ABB RobotStudio station: TCP_Station.rspag

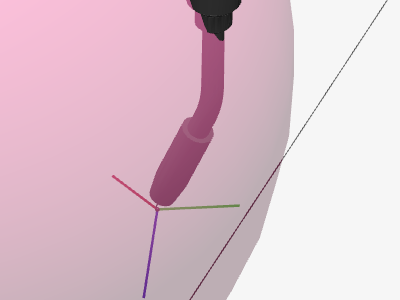
--- station ---
Station TCP_Station (saved by RobotStudio 24.3.10835.0)
Controller IRB2600_12_165, task T_ROB1: task frame (RAPID world) sits at (0, 0, 400) mm in the station
Controller IRB2600_12_165
  mechanical unit ROB_1: IRB2600_12_165_C_01, 6 joints, base frame (0, 0, 0) mm
Layout (positions relative to the parent item):
  - IRB2600_12_165_C_01 [mechanism, from %ABB.RobotStudio.Models.IRB2600%\IRB2600_12_165_C_01.rslib] at (0, 0, 400) mm; joint values [0.0936, 0.2987, 0.0097, 2.8158, -0.9379, -2.8759] (rad or m)
  - Robot Riser Type A_400 mm [part], size 869.6 x 869.6 x 400 mm
  - RA_MTG4000_22 [mechanism, from %ABB.RobotStudio.Models.ArcWelding%\Fronius_Robacta_MTG4000_22deg.rslib] at (1173.49, 88.1, 1305.09) mm, rotated rx -166.47 ry 21.04 rz -178.7 deg
  - WorldTip [part] at (1000, 0, 0) mm, size 600 x 600 x 1000 mm
  - SphereInWobj0 [part] at (1000.44, 0.09, 998.26) mm, size 726.5 x 724 x 729 mm
  - SphereInTool0 [part] at (1173.49, 88.1, 1305.09) mm, rotated rx -166.47 ry 21.04 rz -178.7 deg, size 3.6 x 3.6 x 3.6 mm
Attachment: RA_MTG4000_22 is attached to IRB2600_12_165_C_01 / Link6
Attachment: SphereInTool0 is attached to IRB2600_12_165_C_01 / Link6

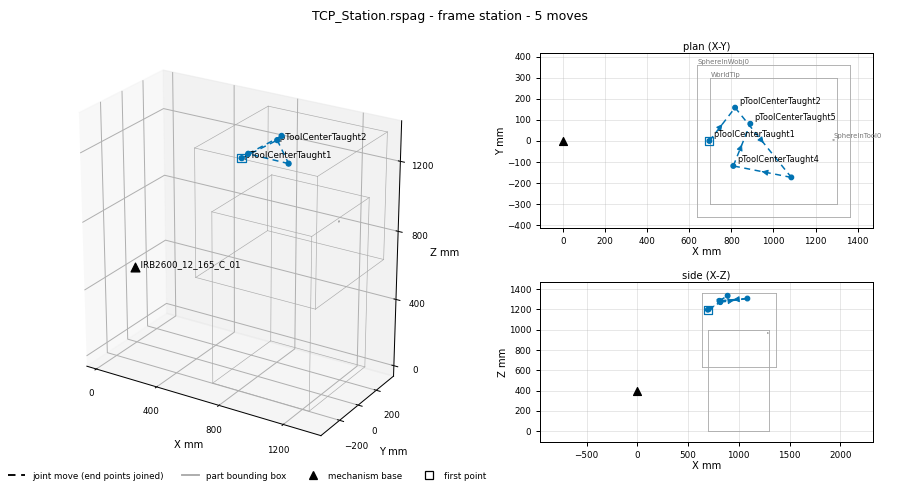
[picture p0: tool path of TCP_Station.rspag in frame station, 5 of 5 moves have a stored position in this frame; points joined in program order, loops and branches not executed]
--- Controller Data/IRB2600_12_165/RAPID/TASK1/PROGMOD/Module1.modx ---
MODULE Module1

!***********************************************************
    !
    ! Module:  Module1
    !
    ! Description:
    !   <Insert description here>
    !
    ! Author: FRFLLOB
    !
    ! Version: 1.0
    !
    !***********************************************************


    !***********************************************************
    !
    ! Procedure main
    !
    !   This is the entry point of your program
    !
!    !***********************************************************
!    PROC main()
!        !Add your code here
!    ENDPROC
ENDMODULE

--- Controller Data/IRB2600_12_165/RAPID/TASK1/PROGMOD/ToolCenterCalculations.modx ---
MODULE ToolCenterCalculations
    ! ------------------------------------------------------------------------------
    ! This module defines a Tool Center calibration process using sphere fitting. If the
    ! number of points taught is 4, the built-in MToolTCPCalib method is used.
    ! The "main" procedure is an example and should be removed to avoid multiple main
    ! definitions. The robtargets are defined using tool0, named pToolCenterTaughtX where
    ! X ranges from 1 to the number of points taught. The module includes procedures
    ! for initializing, calculating the Tool Center Point (TCP), and displaying results.
    ! ------------------------------------------------------------------------------

    ! nNumberPoints defines the number of points used for ToolCenter calibration
    CONST num nNumberPoints:=5; ! EDIT HERE
    VAR robtarget robtargetsArray{nNumberPoints};
    ! Robtargets defined using tool0 pointing at the world fixed tip in wobj0
    ! Names has to be pToolCenterTaughtX where X go from 1 to the number of points taught
    CONST robtarget pToolCenterTaught1:=[[695.487947126,0,797.189508412],[0.500000013,0,0.866025396,0],[0,0,0,0],[9E+09,9E+09,9E+09,9E+09,9E+09,9E+09]];
    CONST robtarget pToolCenterTaught2:=[[817.6949914,158.289988082,871.790822234],[0.272802268,-0.083448092,0.924618094,-0.252382087],[0,1,-2,1],[9E+09,9E+09,9E+09,9E+09,9E+09,9E+09]];
    CONST robtarget pToolCenterTaught3:=[[1084.79999022,-173.063794811,907.667532876],[0.008615643,0.305478727,-0.909287118,-0.282498593],[-1,2,-3,1],[9E+09,9E+09,9E+09,9E+09,9E+09,9E+09]];
    CONST robtarget pToolCenterTaught4:=[[809.124803349,-118.646502119,885.389423002],[0.015910988,-0.85093872,-0.42992302,-0.301357482],[-1,2,-1,1],[9E+09,9E+09,9E+09,9E+09,9E+09,9E+09]];
    CONST robtarget pToolCenterTaught5:=[[889.974092933,81.704160916,935.323503069],[0.182620205,0.01041126,0.976524884,-0.113756831],[0,1,-2,1],[9E+09,9E+09,9E+09,9E+09,9E+09,9E+09]];
    ! CONST robtarget pToolCenterTaughtX:=...; ! EDIT HERE

    PERS pos posArraySphereTool0{nNumberPoints};

    VAR pos posCenterSphereWobj0;
    VAR num nRadiusSphereWobj0;

    VAR pos posToolCenter;
    VAR num nMaxError;
    VAR num nMeanError;

    ! Result:
    TASK PERS tooldata toolToDeterminate:=[TRUE,[[18.6199,-0.147497,364.665],[0.946578,0.191449,0.0562058,0.253336]],[1,[0,0,1],[1,0,0,0],0,0,0]];

    PROC main()
        init;
        calcToolCenter;
        displayResults;
    ERROR
        ExitCycle;
    ENDPROC

    PROC calcError()
        VAR num sum:=0;
        VAR num dist;
        nMeanError:=0;
        nMaxError:=0;

        FOR i FROM 1 TO nNumberPoints DO
            dist:=Distance(posToolCenter,posArraySphereTool0{i});
            sum:=sum+dist;
            nMaxError:=Max(nMaxError,dist);
        ENDFOR
        nMeanError:=sum/nNumberPoints;
    ENDPROC

    PROC calcToolCenter()
        ! MToolTCPCalib is a built-in routine if the number of points taught is 4.
        VAR num max_err;
        VAR num mean_err;
        IF nNumberPoints=4 THEN
            MToolTCPCalib CalcJointT(pToolCenterTaught1,tool0),CalcJointT(pToolCenterTaught2,tool0),CalcJointT(pToolCenterTaught3,tool0),CalcJointT(pToolCenterTaught4,tool0),toolToDeterminate,max_err,mean_err;
            posToolCenter:=toolToDeterminate.tframe.trans;
            nMeanError:=mean_err;
            nMaxError:=max_err;
        ELSE
            ! Calculates the Tool Center Point (ToolCenter) based on sphere fitting
            findSphereInWobj0;
            findSphereInTool0;
            toolToDeterminate.tframe.trans:=posToolCenter;
        ENDIF
    ERROR
        RAISE ;
    ENDPROC

    PROC displayResults()
        TPWrite "ToolCenter Calibration Complete";
        TPWrite "ToolCenter Position: "\pos:=posToolCenter;
        TPWrite "  Max Error: "\num:=nMaxError;
        TPWrite "  Mean Error: "\num:=nMeanError;
    ENDPROC

    PROC findSphereInTool0()
        ! Finds the center and radius of a sphere in the tool frame
        VAR pos posCenterTemp;
        VAR num nRadiusTemp;
        ! Calculate the position of the center of the sphere in the tool frame for every point taught
        FOR i FROM 1 TO nNumberPoints DO
            posArraySphereTool0{i}:=PoseVect(PoseInv([robtargetsArray{i}.trans,robtargetsArray{i}.rot]),posCenterSphereWobj0);
        ENDFOR
        ! Find the sphere created by the points in the tool frame
        FitSphere posArraySphereTool0,posCenterTemp,nRadiusTemp;
        posToolCenter:=posCenterTemp;
        calcError;
    ENDPROC

    PROC findSphereInWobj0()
        ! Finds the center and radius of a sphere in the work object frame
        VAR pos posCenterTemp;
        VAR num nRadiusTemp;
        VAR pos posArraySphereWobj0{nNumberPoints};
        FOR i FROM 1 TO nNumberPoints DO
            posArraySphereWobj0{i}:=robtargetsArray{i}.trans;
        ENDFOR
        FitSphere posArraySphereWobj0,posCenterTemp,nRadiusTemp;
        posCenterSphereWobj0:=posCenterTemp;
        nRadiusSphereWobj0:=nRadiusTemp;
    ERROR
        IF ERRNO=ERR_FIT_TOO_FEW_POINTS THEN
            TPWrite "Error: Too few points to determine the sphere. At least 3 points are required.";
        ELSEIF ERRNO=ERR_FIT_TOO_MANY_POINTS THEN
            TPWrite "Error: Too many points to determine the sphere. Maximum allowed is 100.";
        ELSEIF ERRNO=ERR_FIT_POINTS_IN_LINE THEN
            TPWrite "Error: Incorrect points given. The points must not be in a straight line.";
        ELSE
            TPWrite "An unexpected error occurred in findSphereInWobj0, ERRNO:"\num:=ERRNO;
        ENDIF
        RAISE ;
    ENDPROC

    PROC init()
        TPErase;
        initializeRobTargetsArray;
    ENDPROC

    PROC initializeRobTargetsArray()
        ! Fill the robtargets array with the taught points
        FOR i FROM 1 TO nNumberPoints DO
            GetDataVal "pToolCenterTaught"+ValToStr(i),robtargetsArray{i};
        ENDFOR
    ERROR
        TPWrite "Impossible to initialize the robtargets array:";
        TPWrite "- check the number of points taught,";
        TPWrite "- the consistency with the variable nNumberPoints,";
        TPWrite "- the naming convention pToolCenterTaughtX";
        RAISE ;
    ENDPROC

    PROC syncRS()
        MoveJ pToolCenterTaught1,vmax,fine,tool0;
        MoveJ pToolCenterTaught2,vmax,fine,tool0;
        MoveJ pToolCenterTaught3,vmax,fine,tool0;
        MoveJ pToolCenterTaught4,vmax,fine,tool0;
        MoveJ pToolCenterTaught5,vmax,fine,tool0;
    ENDPROC
ENDMODULE

--- Controller Data/IRB2600_12_165/SYSPAR/EIO.cfg ---
EIO:CFG_1.0:7:0::
#
VIRTUAL_NETWORK:

      -Name "Virtual" -Label "Virtual Device Network"

#CTRL_SIGNATURE:2kwlKDzALXwKJutOOunS4nPoZHdJKPaJW9u0A3DfXbDabHTUop/QpfbvUS3W27GrnjGLWNex2NEpcPv7+bTOLg==

--- Controller Data/IRB2600_12_165/SYSPAR/PROC.cfg ---
PROC:CFG_1.0:7:0::

#CTRL_SIGNATURE:7bhj27i0BeLMM2wKMe22BU7YRfn/9Put1W+rJ4BEeSFKq7o2EtDAOHPMnmvKvl79+M1Z6a/iyijEGw0YvsoC2g==
